FUNCTION_BLOCK SerialLineControl_ADS IMPLEMENTS I_Cyclic, I_SerialLineControl
VAR
	seriallinectrl : SerialLineControlADS := (Timeout := T#5S);
	txComBuffer	   : Tc2_SerialCom.ComBuffer;
	rxComBuffer	   : Tc2_SerialCom.ComBuffer;
END_VAR

METHOD CyclicLogic
seriallinectrl(Connect := TRUE, TxBuffer := txComBuffer, RxBuffer := rxComBuffer);
END_METHOD

PROPERTY rxBuffer : REFERENCE TO combuffer
GET
rxBuffer REF= rxComBuffer;
END_GET
END_PROPERTY

METHOD SetConnectionConfig : BOOL
VAR_INPUT
	ComportSettings : ComSerialConfig;
	NetId			: T_AmsNetId := '';
END_VAR
seriallinectrl.SerialCfg := ComportSettings;
seriallinectrl.NetId	 := NetId;
SetConnectionConfig		 := TRUE;
END_METHOD

PROPERTY txBuffer : REFERENCE TO combuffer
GET
txBuffer REF= txComBuffer;
END_GET
END_PROPERTY

END_FUNCTION_BLOCK

(* stored: Version 1.1.0.1, ProductVersion 3.1.4026.18
   POU SerialLineControl_ADS: Id {ea07a90d-47f5-45b7-afa8-664e72fa7232}, SpecialFunc None
   Method CyclicLogic: Id {30bc274c-02c1-4279-8be4-440759f8f3fe}
   Property rxBuffer: Id {0cedc798-d265-462e-ad66-e3fa206dacc3}
   Get Get: Id {82f93b8f-1d00-4bc1-aada-0b3e795b36a0}
   Method SetConnectionConfig: Id {d19ae4b0-a9c2-4ce5-8102-ff83535335ab}
   Property txBuffer: Id {c09e6bad-f5d8-4750-b6ed-fa9581cc14e1}
   Get Get: Id {b836d6b7-384f-4e8a-b7d1-e66f7771267c} *)
